{attribute 'linkalways'} 
{attribute 'no_explicit_call' := 'This FB is a CLASS and must be accessed using methods or properties'}
{attribute 'enable_dynamic_creation'}
FUNCTION_BLOCK _TcVnPoint3_REAL EXTENDS AliasDatatypeBase
VAR
	localData : TcVnPoint3_REAL;
	activeData : REFERENCE TO TcVnPoint3_REAL REF= localData;
	aliasBaseDatatype : _TcVnVector3_REAL;
END_VAR

PROPERTY PUBLIC Address : PVOID
GET
Address := ADR(activeData);
END_GET
END_PROPERTY

METHOD PUBLIC ClearReference
VAR_INPUT
END_VAR
activeData REF= localData;
SetBaseDatatypeReference();
END_METHOD

METHOD PUBLIC Clone : I_Datatype
VAR
    pClone : POINTER TO _TcVnPoint3_REAL;
END_VAR
pClone := __NEW(_TcVnPoint3_REAL);
Clone := pClone^;
END_METHOD

METHOD FB_init : BOOL
VAR_INPUT
	bInitRetains : BOOL; // if TRUE, the retain variables are initialized (warm start / cold start)
	bInCopyCode : BOOL;  // if TRUE, the instance afterwards gets moved into the copy code (online change)
	//InitialValue : <type>; // if possible, not all values can be initialized
END_VAR
//localData := InitialValue; // if possible, not all values can be initialized
SetBaseDatatypeReference();
AddBaseDatatype(aliasBaseDatatype);
END_METHOD

PROPERTY PUBLIC Identifier : T_MAXSTRING
GET
Identifier := 'TcVnPoint3_REAL';
END_GET
END_PROPERTY

METHOD PUBLIC MakeReferenceTo
VAR_INPUT
	ReferenceTarget : REFERENCE TO TcVnPoint3_REAL;
END_VAR
activeData REF= ReferenceTarget;
SetBaseDatatypeReference();
END_METHOD

METHOD PROTECTED SetBaseDatatypeReference
VAR_INPUT
END_VAR
aliasBaseDatatype.MakeReferenceTo(activeData);
END_METHOD

PROPERTY PUBLIC Size : UDINT
GET
Size := SIZEOF(activeData);
END_GET
END_PROPERTY

METHOD TryMakeReferenceTo : BOOL
VAR_INPUT
	Target : I_Datatype;
END_VAR
VAR
	pTargetData : POINTER TO TcVnPoint3_REAL;
END_VAR
IF NOT IsEquivalentTo(Target) THEN
	RETURN;
END_IF

pTargetData := Target.Address;
activeData REF= pTargetData^;
SetBaseDatatypeReference();
TryMakeReferenceTo := TRUE;
END_METHOD

PROPERTY PUBLIC Value : REFERENCE TO TcVnPoint3_REAL
GET
Value REF= activeData;
END_GET
END_PROPERTY

END_FUNCTION_BLOCK

(* stored: Version 1.1.0.1, ProductVersion 3.1.4024.13
   POU _TcVnPoint3_REAL: Id {7e0b2149-5d4c-0dc0-179e-3bcb8d62b486}, SpecialFunc None
   Folder Core: Id {af40a993-02e5-0d62-3a15-e83a8d0089cb}
   Folder Protected: Id {3fbfa86e-44a3-0531-1771-b40b77e80f73}
   Folder Customize: Id {2af7a419-fb88-02a8-04f9-fa30b1d3c373}
   Folder Constructor: Id {3285c11c-514e-07cd-07d0-74d05914385b}
   Property Address: Id {b66c3166-81fb-0886-1515-5913a3721e02}
   Get Get: Id {8135928f-05bb-06fc-346c-6429ae7c612f}
   Method ClearReference: Id {9207bf0d-085c-0d77-189f-8041c866844d}
   Method Clone: Id {c0b3e315-79fd-0885-0139-c6671e156064}
   Method FB_init: Id {1bdd922a-6269-05f3-1bb1-a02c3a294299}
   Property Identifier: Id {565e5c8a-7957-07bf-0a84-259bd7a6a14e}
   Get Get: Id {23f6dcb3-8948-0bbe-1572-8c9c0c4a40d1}
   Method MakeReferenceTo: Id {eeefde4d-80e0-0b0a-2132-abbeea1c6ade}
   Method SetBaseDatatypeReference: Id {ee0b7208-8804-02b5-0251-b800ddf47de8}
   Property Size: Id {62e2d3a7-7ab0-0e82-21b4-7d8c33ec60ab}
   Get Get: Id {fb20ee73-1cf0-0529-1a3d-04545c6ebaef}
   Method TryMakeReferenceTo: Id {c1a75e02-be3b-0027-2a1a-e4a9e998f00a}
   Property Value: Id {238812b6-e4bb-0647-0c6e-b44667b26950}
   Get Get: Id {15a6b348-2250-0ce4-0149-6caec6ab7216} *)
